// TwinCAT 3 PLC project UR5_Test
// ProgramVersion: 3.1.4026.10
// libraries:
//   Tc2_Standard, * (Beckhoff Automation GmbH)
//   Tc2_System, * (Beckhoff Automation GmbH)
//   Tc2_TcpIp, * (Beckhoff Automation GmbH)
//   Tc2_Utilities, * (Beckhoff Automation GmbH)
// project tree:
//   DUTs/ DATA.TcDUT, DATA_R.TcDUT, RealTimeData.TcDUT, Variablen.TcDUT
//   / PlcTask.TcTTO
//   POUs/ Kommunikation_Client.TcPOU, Kommunikation_Server.TcPOU, MAIN.TcPOU
// real-time tasks:
//   TASK PlcTask: cycle T#10ms, priority 20, ADS port 350
// I/O:
//   DEVICE Gerät 1 (RT-Ethernet Adapter)

CONFIGURATION UR5_Test
    RESOURCE PLC ON TwinCAT3
        TASK PlcTask(INTERVAL := T#10ms, PRIORITY := 20);
        PROGRAM MAIN WITH PlcTask : MAIN;
    END_RESOURCE
END_CONFIGURATION

// ---- DUTs/DATA.TcDUT
TYPE DATA :
UNION
  stTest : STRING;
  arTest : ARRAY[0..255] OF BYTE;
END_UNION
END_TYPE

// ---- DUTs/DATA_R.TcDUT
TYPE DATA_R :
UNION
  arrByte :		 ARRAY[0..3] OF BYTE;
  rReal		 	:REAL;
END_UNION
END_TYPE

// ---- DUTs/RealTimeData.TcDUT
TYPE RealTimeData :
STRUCT
	messageSize 				: ARRAY[0..3] OF BYTE;
	timestamp 					: ARRAY[0..7] OF BYTE;
	qTarget 					: ARRAY[0..47] OF BYTE;
	qdTarget 					: ARRAY[0..47] OF BYTE;
	qddTarget 					: ARRAY[0..47] OF BYTE;
	iTarget 					: ARRAY[0..47] OF BYTE;
	mTarget 					: ARRAY[0..47] OF BYTE;
	qActual 					: ARRAY[0..47] OF BYTE;
	qdActual 					: ARRAY[0..47] OF BYTE;
	iActual 					: ARRAY[0..47] OF BYTE;
	toolAccelerometerValues 	: ARRAY[0..23] OF BYTE;
	unused 						: ARRAY[0..119] OF BYTE;
	tcpForce 					: ARRAY[0..47] OF BYTE;
	toolVector 					: ARRAY[0..47] OF BYTE;
	tcpSpeed 					: ARRAY[0..47] OF BYTE;
	digitalInputBits 			: ARRAY[0..7] OF BYTE;
END_STRUCT
END_TYPE

// ---- DUTs/Variablen.TcDUT
TYPE Variablen :
STRUCT
	q1		: ARRAY[0..7] OF BYTE;
	q2		: ARRAY[0..7] OF BYTE;
	q3		: ARRAY[0..7] OF BYTE;
	q4		: ARRAY[0..7] OF BYTE;
	q5		: ARRAY[0..7] OF BYTE;
	q6		: ARRAY[0..7] OF Byte;
END_STRUCT
END_TYPE

// ---- POUs/MAIN.TcPOU
PROGRAM MAIN
VAR
	remotePort		:UDINT := 30003;
	remoteHost		:T_IPv4Addr := '192.168.50.100';
	
	data 			:T_MaxString := 'get_actual_joint_positions()';
	receivedData	:RealTimeData;
	testR			:DATA_R;
	
	rMyRealValue	:INT;
	pReal 			:POINTER TO INT;
	testArray1:		ARRAY[0..3] OF BYTE := [0, 0, 3, 44];
	testArray2:		ARRAY[0..3] OF BYTE := [44, 3, 0, 0];

	stTest			:DATA; 
	test3			:T_MaxString := 'movej([0,1.57,-1.57,3.14,-1.57,1.57],a=0.2,v=0.2,t=0,r=0)\n';
	
	actualLength : UDINT;                  // Tatsächliche Länge des Strings
    i            : UDINT;                  // Schleifenvariabl
	byteArray    : POINTER TO ARRAY[0..255] OF BYTE;
	newArray    : POINTER TO ARRAY[0..51] OF BYTE;
END_VAR

VAR_INPUT
	socket				:T_HSOCKET;
	hListener_OUT 		:T_HSOCKET;
	hListener_IN 		:T_HSOCKET;
END_VAR



Kommunikation_Server();
Kommunikation_Client();

//stTest.stTest := 'force()';
stTest.stTest := 'force()';

actualLength := LEN(stTest.stTest);
stTest.arTest[actualLength] := 10;

testR.arrByte := receivedData.messageSize;
//pReal := ADR(receivedData.messageSize);
//rMyRealValue := pReal^;

pReal := ADR(testArray2);
rMyRealValue := pReal^;


hListener_IN.handle := hListener_OUT.handle;
hListener_IN.localAddr.sAddr := '192.168.50.10';
hListener_IN.localAddr.nPort := 53828;
hListener_IN.remoteAddr.sAddr := remoteHost;
hListener_IN.remoteAddr.nPort := remotePort;

END_PROGRAM

// ---- POUs/Kommunikation_Server.TcPOU
PROGRAM Kommunikation_Server
VAR
	Connect			:FB_ServerClientConnection;
	Connect_Local	:FB_SocketConnect;
	Send			:FB_SocketSend;
	Receive			:FB_SocketReceive;
	hServer			:T_HSERVER;
	
	sSrvNetID : T_AmsNetID := '';
	sLocalHost : STRING(15) := '147.87.210.78';
	nLocalPort : UDINT := 21;
	nMode : DWORD := LISTEN_MODE_CLOSEALL (* OR CONNECT_MODE_ENABLEDBG*);
	bEnable : BOOL := TRUE;
	
	eMode       : E_SocketAcceptMode := eACCEPT_ALL;
    sRemoteHost : T_IPv4Addr := '192.168.50.100';
    nRemotePort : UDINT := 30002;
    tReconnect  : TIME := T#5S;
	
END_VAR

VAR_INPUT
	
	
	
END_VAR

F_CreateServerHnd(sSrvNetID := sSrvNetID, sLocalHost := sLocalHost, nLocalPort := nLocalPort, nMode := nMode, bEnable := bEnable, hServer := hServer);
Connect(
    hServer := hServer,
    eMode := eMode,
    sRemoteHost := sRemoteHost,
    nRemotePort := nRemotePort,
    bEnable := bEnable,
    tReconnect := tReconnect); // FB_ServerClientConnection
Send(hSocket := MAIN.socket, cbLen := SIZEOF(MAIN.data), pSrc := ADR(MAIN.data)); // FB_SocketSend
Receive(hSocket := MAIN.socket); // FB_SocketReceive

END_PROGRAM

// ---- POUs/Kommunikation_Client.TcPOU
PROGRAM Kommunikation_Client
VAR
	Connect			:FB_SocketConnect;
	Send			:FB_SocketSend;
	Receive 		:FB_SocketReceive;
	CloseAll		:FB_SocketCloseAll;
	
	sSrvNetId   : T_AmsNetId := '';
    sRemoteHost : T_IPv4Addr := '192.168.50.100';
    nRemotePort : UDINT := 30003;
    bConnect    : BOOL;
    tTimeout    : TIME := T#45S;(*!!!*)
	bSend		:BOOL;
	bReceive	:BOOL;
	
	hSocket    : T_HSOCKET;
	
	{attribute 'TcEncoding':='UTF-8'}
	//test		:T_MaxString := 'movej([0,1.57,-1.57,3.14,-1.57,1.57],a=0.2,v=0.2,t=0,r=0)/n'; 
	test		:T_MaxString := 'force()'; 
	{attribute 'TcEncoding':='UTF-8'}
	Test2		:STRING := 'socket_send_byte(10)'; 
	test6		:ARRAY[0..7] OF BYTE := [102,111,114,99,101,40,41,10];

	
END_VAR

Send(
    sSrvNetId := sSrvNetId,
    hSocket := hSocket,
    cbLen := LEN( MAIN.stTest.stTest),
    pSrc := ADR(MAIN.stTest.arTest),
    bExecute := bSend); // FB_SocketSend
Connect(
    sSrvNetId := sSrvNetId,
    sRemoteHost := sRemoteHost,
    nRemotePort := nRemotePort,
    bExecute := bConnect,
    tTimeout := tTimeout); // FB_SocketConnect
hSocket := Connect.hSocket;
CloseAll(sSrvNetId := sSrvNetId); // FB_SocketCloseAll
Receive(
    sSrvNetId := sSrvNetId,
    hSocket := hSocket,
    cbLen := SIZEOF(Main.receivedData),
    pDest := ADR(Main.receivedData),
    bExecute := bReceive); // FB_SocketReceive

END_PROGRAM
